// Mitsubishi GX Works2 project: 250916_A+A-B+B-C+C- 반복   PLC: Q02U

PROGRAM MAIN
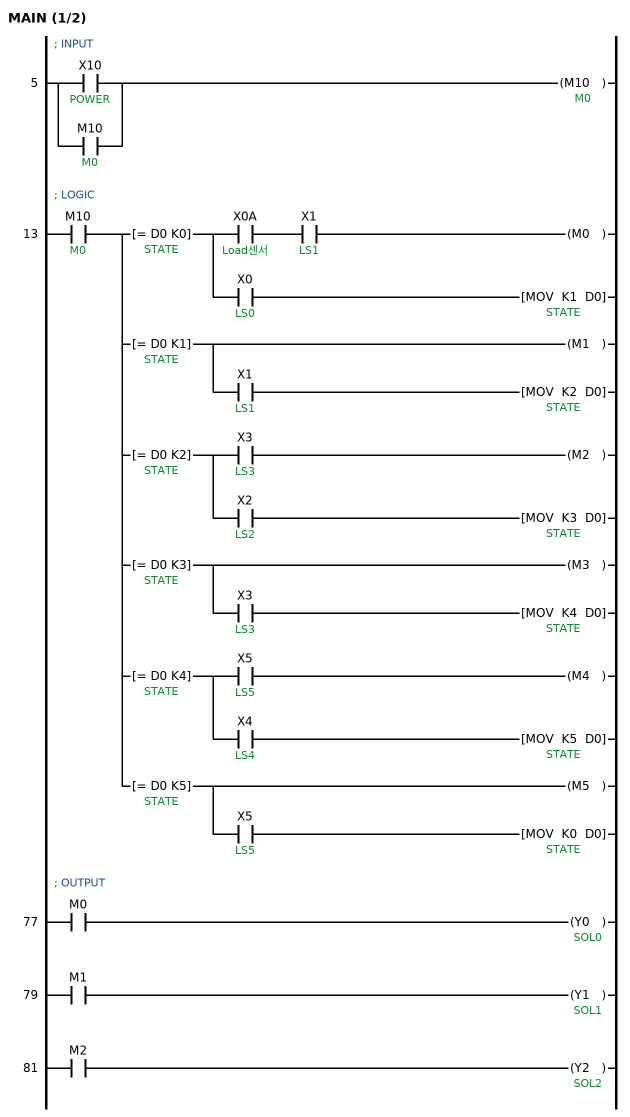
; INPUT
5     LD      X10  ; POWER
      OR      M10  ; M0
      OUT     M10  ; M0
; LOGIC
13    LD      M10  ; M0
      MPS
      AND=    D0 K0  ; STATE
      MPS
      AND     X0A  ; Load센서
      AND     X1  ; LS1
      OUT     M0
      MPP
      AND     X0  ; LS0
      MOV     K1 D0
      MRD
      AND=    D0 K1  ; STATE
      OUT     M1
      AND     X1  ; LS1
      MOV     K2 D0
      MRD
      AND=    D0 K2  ; STATE
      MPS
      AND     X3  ; LS3
      OUT     M2
      MPP
      AND     X2  ; LS2
      MOV     K3 D0
      MRD
      AND=    D0 K3  ; STATE
      OUT     M3
      AND     X3  ; LS3
      MOV     K4 D0
      MRD
      AND=    D0 K4  ; STATE
      MPS
      AND     X5  ; LS5
      OUT     M4
      MPP
      AND     X4  ; LS4
      MOV     K5 D0
      MPP
      AND=    D0 K5  ; STATE
      OUT     M5
      AND     X5  ; LS5
      MOV     K0 D0
; OUTPUT
77    LD      M0
      OUT     Y0  ; SOL0
79    LD      M1
      OUT     Y1  ; SOL1
81    LD      M2
      OUT     Y2  ; SOL2
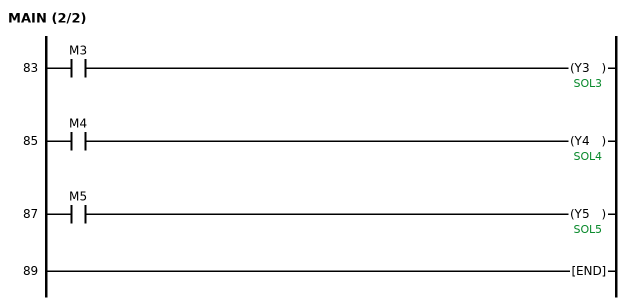
83    LD      M3
      OUT     Y3  ; SOL3
85    LD      M4
      OUT     Y4  ; SOL4
87    LD      M5
      OUT     Y5  ; SOL5
89    END
END_PROGRAM

// device comments not shown above
X6  ; LS6
X7  ; LS7
X8  ; 근접센서
X9  ; 금속센서
Y6  ; SOL6
Y7  ; SOL7
Y8  ; CONV ON/OFF
Y9  ; CONV CW
Y0A  ; CONV CCW
Y0B  ; RED LAMP
Y0C  ; YELLOW LAMP
Y0D  ; GREEN LAMP
